// TIA Portal V20 export
TYPE "UDT_FuellstandStoe"
   STRUCT
      MESS_DB_STOE : Bool;
      xRes0 : Bool;
      xRes1 : Bool;
      xRes2 : Bool;
      xRes3 : Bool;
      xRes4 : Bool;
      xRes5 : Bool;
      xRes6 : Bool;
      bRes1 : Byte;
   END_STRUCT;
END_TYPE
